(* IEC 61131-3 sources: volt/packages/volt-lsp-iec/test-corpus/pro2193/Device/Plc Logic/Application/99 Library/Functions/Implicit Check Functions, 10 files *)

(* ---- CheckBounds.pou ---- *)
// Implicitly generated code : DO NOT EDIT
FUNCTION CheckBounds : DINT
VAR_INPUT
	index, lower, upper : DINT;
END_VAR

%LANGUAGE ST
%CLASS CHECK CheckBounds
IF index >= lower AND index <= upper THEN
	CheckBounds := index;
ELSE
	LogPlc.Fatal(CONCAT7(	'CheckBounds Error. Act index ',
							TO_STRING(index),
							' not in range [',
							TO_STRING(lower),
							', ',
							TO_STRING(upper),
							']'));

	CheckBounds := LIMIT(lower, index, upper);

	{IF defined (IsSimulationMode)}
		ThrowException('RtsExceptions.RTSEXCPT_ARRAYBOUNDS');
	{END_IF}

	IF GlobalVars.CheckBoundFunctionsThrowExceptions THEN
		ThrowException('RtsExceptions.RTSEXCPT_ARRAYBOUNDS');
	END_IF
END_IF

END_FUNCTION

(* ---- CheckDivDInt.pou ---- *)
// Implicitly generated code : DO NOT EDIT
FUNCTION CheckDivDInt : DINT
VAR_INPUT
	divisor		: DINT;
END_VAR

%LANGUAGE ST
%CLASS CHECK CheckDivInt32
IF divisor <> 0 THEN
	CheckDivDInt := divisor;
ELSE
	LogPlc.Fatal('CheckDivDINT Error; Do not divide by 0!');

	CheckDivDInt := 1;

	{IF defined (IsSimulationMode)}
		ThrowException('RtsExceptions.RTSEXCPT_DIVIDEBYZERO');
	{END_IF}

	IF GlobalVars.CheckBoundFunctionsThrowExceptions THEN
		ThrowException('RtsExceptions.RTSEXCPT_DIVIDEBYZERO');
	END_IF
END_IF

END_FUNCTION

(* ---- CheckDivLInt.pou ---- *)
// Implicitly generated code : DO NOT EDIT
FUNCTION CheckDivLInt : LINT
VAR_INPUT
	divisor		: LINT;
END_VAR

%LANGUAGE ST
%CLASS CHECK CheckDivInt64
IF divisor <> 0 THEN
	CheckDivLInt := divisor;
ELSE
	LogPlc.Fatal('CheckDivLINT Error; Do not divide by 0!');

	CheckDivLInt := 1;

	{IF defined (IsSimulationMode)}
		ThrowException('RtsExceptions.RTSEXCPT_DIVIDEBYZERO');
	{END_IF}

	IF GlobalVars.CheckBoundFunctionsThrowExceptions THEN
		ThrowException('RtsExceptions.RTSEXCPT_DIVIDEBYZERO');
	END_IF
END_IF

END_FUNCTION

(* ---- CheckDivLReal.pou ---- *)
// Implicitly generated code : DO NOT EDIT
FUNCTION CheckDivLReal : LREAL
VAR_INPUT
	divisor		: LREAL;
END_VAR

%LANGUAGE ST
%CLASS CHECK CheckDivReal64
IF divisor <> 0 THEN
	CheckDivLReal := divisor;
ELSE
	LogPlc.Fatal('CheckDivLReal Error; Do not divide by 0!');

	CheckDivLReal := 1;

	{IF defined (IsSimulationMode)}
		ThrowException('RtsExceptions.RTSEXCPT_DIVIDEBYZERO');
	{END_IF}

	IF GlobalVars.CheckBoundFunctionsThrowExceptions THEN
		ThrowException('RtsExceptions.RTSEXCPT_DIVIDEBYZERO');
	END_IF
END_IF

END_FUNCTION

(* ---- CheckDivReal.pou ---- *)
// Implicitly generated code : DO NOT EDIT
FUNCTION CheckDivReal : REAL
VAR_INPUT
	divisor		: REAL;
END_VAR

%LANGUAGE ST
%CLASS CHECK CheckDivReal32
IF divisor <> 0 THEN
	CheckDivReal := divisor;
ELSE
	LogPlc.Fatal('CheckDivReal Error; Do not divide by 0!');

	CheckDivReal := 1;

	{IF defined (IsSimulationMode)}
		ThrowException('RtsExceptions.RTSEXCPT_DIVIDEBYZERO');
	{END_IF}

	IF GlobalVars.CheckBoundFunctionsThrowExceptions THEN
		ThrowException('RtsExceptions.RTSEXCPT_DIVIDEBYZERO');
	END_IF
END_IF

END_FUNCTION

(* ---- CheckLRangeSigned.pou ---- *)
// Implicitly generated code : DO NOT EDIT
FUNCTION CheckLRangeSigned : LINT
VAR_INPUT
	value, lower, upper : LINT;
END_VAR

%LANGUAGE ST
%CLASS CHECK CheckLRangeSigned
IF value >= lower AND value <= upper THEN
	CheckLRangeSigned := value;
ELSE
	LogPlc.Fatal(CONCAT7(	'CheckLRangeSigned Error. Act value ',
							TO_STRING(value),
							' not in range (',
							TO_STRING(lower),
							', ',
							TO_STRING(upper),
							')'));

	CheckLRangeSigned := LIMIT(lower, value, upper);

	{IF defined (IsSimulationMode)}
		ThrowException('RtsExceptions.RTSEXCPT_MISALIGNMENT');
	{END_IF}

	IF GlobalVars.CheckBoundFunctionsThrowExceptions THEN
		ThrowException('RtsExceptions.RTSEXCPT_MISALIGNMENT');
	END_IF
END_IF

END_FUNCTION

(* ---- CheckLRangeUnsigned.pou ---- *)
// Implicitly generated code : DO NOT EDIT
FUNCTION CheckLRangeUnsigned : ULINT
VAR_INPUT
	value, lower, upper : ULINT;
END_VAR

%LANGUAGE ST
%CLASS CHECK CheckLRangeUnsigned
IF value >= lower AND value <= upper THEN
	CheckLRangeUnsigned := value;
ELSE
	LogPlc.Fatal(CONCAT7(	'CheckLRangeUnsigned Error. Act value ',
							TO_STRING(value),
							' not in range (',
							TO_STRING(lower),
							', ',
							TO_STRING(upper),
							')'));

	CheckLRangeUnsigned := LIMIT(lower, value, upper);

	{IF defined (IsSimulationMode)}
		ThrowException('RtsExceptions.RTSEXCPT_MISALIGNMENT');
	{END_IF}

	IF GlobalVars.CheckBoundFunctionsThrowExceptions THEN
		ThrowException('RtsExceptions.RTSEXCPT_MISALIGNMENT');
	END_IF
END_IF

END_FUNCTION

(* ---- CheckPointer.pou ---- *)
// Implicitly generated code : DO NOT EDIT
FUNCTION CheckPointer : POINTER TO BYTE
VAR_INPUT
	ptToTest	: POINTER TO BYTE;	// Destination address of the pointer
	iSize		: DINT;				// Size of the type the pointer points to. (e.g: 20 for POINTER TO ARRAY[0..9] OF INT)
	iGran		: DINT;				// Granularity of the pointer access. This is the size of the biggest non-structured data type in the type the pointer points to. (e.g: 2 for POINTER TO ARRAY[0..9] OF INT)
	bWrite		: BOOL;				// Indicates read or write access. TRUE = write access.
END_VAR

%LANGUAGE ST
%CLASS CHECK CheckPointer
%EXCLUDE_FROM_BUILD
// No standard way of implementation. Fill your own code here
CheckPointer := ptToTest;

// THIS FUNCTION IS DISABLED BECAUSE WE DON'T USE IT.
// IT IS CALLED MANY MANY TIMES AND IT AFFECTS PERFORMANCE

END_FUNCTION

(* ---- CheckRangeSigned.pou ---- *)
// Implicitly generated code : DO NOT EDIT
FUNCTION CheckRangeSigned : DINT
VAR_INPUT
	value, lower, upper : DINT;
END_VAR

%LANGUAGE ST
%CLASS CHECK CheckRangeSigned
IF value >= lower AND value <= upper THEN
	CheckRangeSigned := value;
ELSE
	LogPlc.Fatal(CONCAT7(	'CheckRangeSigned Error. Act value ',
							TO_STRING(value),
							' not in range (',
							TO_STRING(lower),
							', ',
							TO_STRING(upper),
							')'));

	CheckRangeSigned := LIMIT(lower, value, upper);

	{IF defined (IsSimulationMode)}
		ThrowException('RtsExceptions.RTSEXCPT_MISALIGNMENT');
	{END_IF}

	IF GlobalVars.CheckBoundFunctionsThrowExceptions THEN
		ThrowException('RtsExceptions.RTSEXCPT_MISALIGNMENT');
	END_IF
END_IF

END_FUNCTION

(* ---- CheckRangeUnsigned.pou ---- *)
// Implicitly generated code : DO NOT EDIT
FUNCTION CheckRangeUnsigned : UDINT
VAR_INPUT
	value, lower, upper : UDINT;
END_VAR

%LANGUAGE ST
%CLASS CHECK CheckRangeUnsigned
IF value >= lower AND value <= upper THEN
	CheckRangeUnsigned := value;
ELSE
	LogPlc.Fatal(CONCAT7(	'CheckRangeUnsigned Error. Act value ',
							TO_STRING(value),
							' not in range (',
							TO_STRING(lower),
							', ',
							TO_STRING(upper),
							')'));

	CheckRangeUnsigned := LIMIT(lower, value, upper);

	{IF defined (IsSimulationMode)}
		ThrowException('RtsExceptions.RTSEXCPT_MISALIGNMENT');
	{END_IF}

	IF GlobalVars.CheckBoundFunctionsThrowExceptions THEN
		ThrowException('RtsExceptions.RTSEXCPT_MISALIGNMENT');
	END_IF
END_IF

END_FUNCTION
